Staubli VAL3: iRack3.pgx

public program iRack3(num& nNum[] (dimensions=1))
begin
  nNum=dioGet(iRack3)
end
